Staubli VAL3: VAL3help_example.dtx

mdesc mNomSpeed
string sInput
string sOutput
string sPrompt
num nRet
bool bExit
